{attribute addProperty BoxType "AX8620-0000-0026"}
{attribute addProperty Id "StatuswordAT %I*Statusword_3B58AC51162"}
{attribute addProperty CRC "854043290"}
{attribute addProperty SizeInBites "16"}
{attribute addProperty SizeInBytes "2"}
TYPE PSM_Statusword_32E7AA9A :
STRUCT
	{attribute addProperty Name "Statusword"}
	Statusword AT %I* : Statusword_3B58AC51;
END_STRUCT
END_TYPE

(* stored: Version 1.2.0.0, ProductVersion 3.1.4024.9
   DUT PSM_Statusword_32E7AA9A: Id {8aee44fc-4a2b-4f86-b4c5-58f2d11f126f} *)
